// Mitsubishi GX Works2 project: Bread   PLC: FX3G

// global labels: Global1
VAR_GLOBAL
  Emergency AT X007 : BOOL;
  InputSpice AT M4 : BOOL;
  InputOil AT M3 : BOOL;
  InputWater AT M2 : BOOL;
  InputShmarim AT M1 : BOOL;
  InputYeast AT M1 : BOOL;
  InputFlour AT M0 : BOOL;
  StateEmergency AT M100 : BOOL;
  ReadyToStart AT Y000 : BOOL;
  StartDay AT X010 : BOOL;
  DayInProgress AT Y010 : BOOL;
  GetInput AT X000 : BOOL;
  AnalogInput1 AT D8280 : INT;
  FlourInStock AT D1101 : REAL;
END_VAR
VAR_GLOBAL CONSTANT
  Flour_Const : REAL := 100;
END_VAR
VAR_GLOBAL
  YeastInStock AT D1103 : REAL;
END_VAR
VAR_GLOBAL CONSTANT
  YeastRatio_Constant : REAL := 0.2;
END_VAR
VAR_GLOBAL
  WaterInStock AT D1105 : REAL;
END_VAR
VAR_GLOBAL CONSTANT
  WatertRatio_Constant : REAL := 0.5;
END_VAR
VAR_GLOBAL
  OilInStock AT D1107 : REAL;
END_VAR
VAR_GLOBAL CONSTANT
  OilRatio_Constant : REAL := 0.3;
END_VAR
VAR_GLOBAL
  SpiceInStock AT D1109 : REAL;
END_VAR
VAR_GLOBAL CONSTANT
  SpiceRatio_Constant : REAL := 0.1;
  Zero_Constant : REAL;
END_VAR
VAR_GLOBAL
  Lisha AT X001 : BOOL;
  Fiktivy AT M200 : BOOL;
  RealNura AT TC1 : BOOL;
END_VAR
VAR_GLOBAL CONSTANT
  mili_900 : INT := 4;
END_VAR
VAR_GLOBAL
  RealNuraTime AT TS1 : BOOL;
  FiktivylNura AT TC2 : BOOL;
END_VAR
VAR_GLOBAL CONSTANT
  mili_100 : INT := 1;
END_VAR
VAR_GLOBAL
  FiktivyNuraTime AT TS2 : BOOL;
  Fiktivy1 AT M300 : BOOL;
  NuraY0 AT M250 : BOOL;
  NuraDay AT M240 : BOOL;
  Emergency_ThreeSeconds AT TC3 : BOOL;
END_VAR
VAR_GLOBAL CONSTANT
  ThreeSeconds : INT := 30;
END_VAR
VAR_GLOBAL
  Emergency_ThreeSeconds_Time AT TS3 : BOOL;
END_VAR
VAR_GLOBAL CONSTANT
  mili_400 : INT := 4;
END_VAR
VAR_GLOBAL
  StartPrepare AT X002 : BOOL;
  Prepare_C AT TC30 : BOOL;
END_VAR
VAR_GLOBAL CONSTANT
  Prepare_milli : INT := 30;
END_VAR
VAR_GLOBAL
  StatePrepare AT M10 : BOOL;
  Prepare_Timer AT TS30 : BOOL;
  PrepareNura AT Y005 : BOOL;
  FinishPrepare AT M11 : BOOL;
  Flour_Mearbel AT D2101 : REAL;
  Yeast_Mearbel AT D2103 : REAL;
END_VAR
VAR_GLOBAL CONSTANT
  Yeast_Const : REAL := 20;
END_VAR
VAR_GLOBAL
  Flour_Meychal AT D2101 : REAL;
  Yeast_Meychal AT D2103 : REAL;
  Water_Meychal AT D2105 : REAL;
  Oil_Meychal AT D2107 : REAL;
END_VAR
VAR_GLOBAL CONSTANT
  Water_Const : REAL := 50;
  Oil_Const : REAL := 30;
  Spice_Const : REAL := 10;
END_VAR
VAR_GLOBAL
  Spice_Meychal AT D2109 : REAL;
  LishaNura AT Y001 : BOOL;
  Spice_Stock AT D1109 : REAL;
  StartHatfahaCount AT CC0 : BOOL;
END_VAR
VAR_GLOBAL CONSTANT
  count2 : INT := 2;
END_VAR
VAR_GLOBAL
  StartHatfaha AT CS0 : BOOL;
  FakeNuraY1 AT M252 : BOOL;
  NuraY2 AT Y002 : BOOL;
  NuraY3 AT Y003 : BOOL;
  Y2NuraTime AT TS10 : BOOL;
  Y3NuraTime AT TS20 : BOOL;
  Hatfaha_ThreeSeconds_Time AT TS80 : BOOL;
  HivHov AT M280 : BOOL;
  HivHovY2 AT TC10 : BOOL;
  HivHovY3 AT TC20 : BOOL;
  Hatfaha_ThreeSeconds AT TC80 : BOOL;
  StartHivHov AT M80 : BOOL;
  Hatfaha_Tavnit AT D4101 : REAL;
END_VAR
VAR_GLOBAL CONSTANT
  Batzekr_Const : REAL := 210;
  Batzek_Const : REAL := 210;
  Afia_time_const : WORD := 40;
END_VAR
VAR_GLOBAL
  NuraY4 AT TC90 : BOOL;
  Hatfaha AT X011 : BOOL;
  Lisha_mearbelNEW AT D3101 : REAL;
  Afia_done AT TS90 : BOOL;
  NuraAfiaY4 AT Y004 : BOOL;
  bdika AT X005 : BOOL;
  bdikanura AT Y011 : BOOL;
  end_hatfaha AT M244 : BOOL;
  StartQA AT X003 : BOOL;
  QA_input AT D5101 : REAL;
END_VAR
VAR_GLOBAL CONSTANT
  QA_const_1 : INT := 400;
  QA_const_5 : INT := 2000;
END_VAR
VAR_GLOBAL
  QA_Success AT M197 : BOOL;
  NuraY6 AT TC95 : BOOL;
END_VAR
VAR_GLOBAL CONSTANT
  shelf_tranfer_time : WORD := 50;
END_VAR
VAR_GLOBAL
  Shelf_transfer_done AT TS95 : BOOL;
  NuraY5 AT Y005 : BOOL;
END_VAR
VAR_GLOBAL CONSTANT
  count_QA_CONST : INT := 2;
END_VAR
VAR_GLOBAL
  count_QA AT CC2 : BOOL;
  count_QA_done AT CS2 : BOOL;
  Afia_tavnit AT D6101 : REAL;
  Fiktivi_QA_succes AT M325 : BOOL;
  Bread_shelf AT D7101 : REAL;
  Greater_than1 AT M222 : BOOL;
  Less_than5 AT M223 : BOOL;
  QA_Success_NuraY6 AT Y006 : BOOL;
  Input_saved AT M127 : BOOL;
  AnalogInput2 AT D8281 : INT;
  AnalogOutput AT D8201 : INT;
  Ingridients_check AT M255 : BOOL;
  AnalogOutputnEW AT D8201 : INT;
  StartHatfaha_current AT CN0 : INT;
  count_QA_current AT CN2 : INT;
END_VAR
VAR_GLOBAL CONSTANT
  Zero_Constant_Word : INT;
END_VAR
VAR_GLOBAL
  Ge_success AT M190 : BOOL;
  Le_success AT M191 : BOOL;
  checkIngridients AT M321 : BOOL;
END_VAR

// task Task_01 (event TRUE, interval 0, priority 31): POU_01

PROGRAM POU_01
VAR
  Lisha_mearbel : REAL;
END_VAR
(* structured ladder/FBD written out as ST: instructions are called as NAME(EN, inputs, outputs); _pN, _eN, _tN stand for wires *)
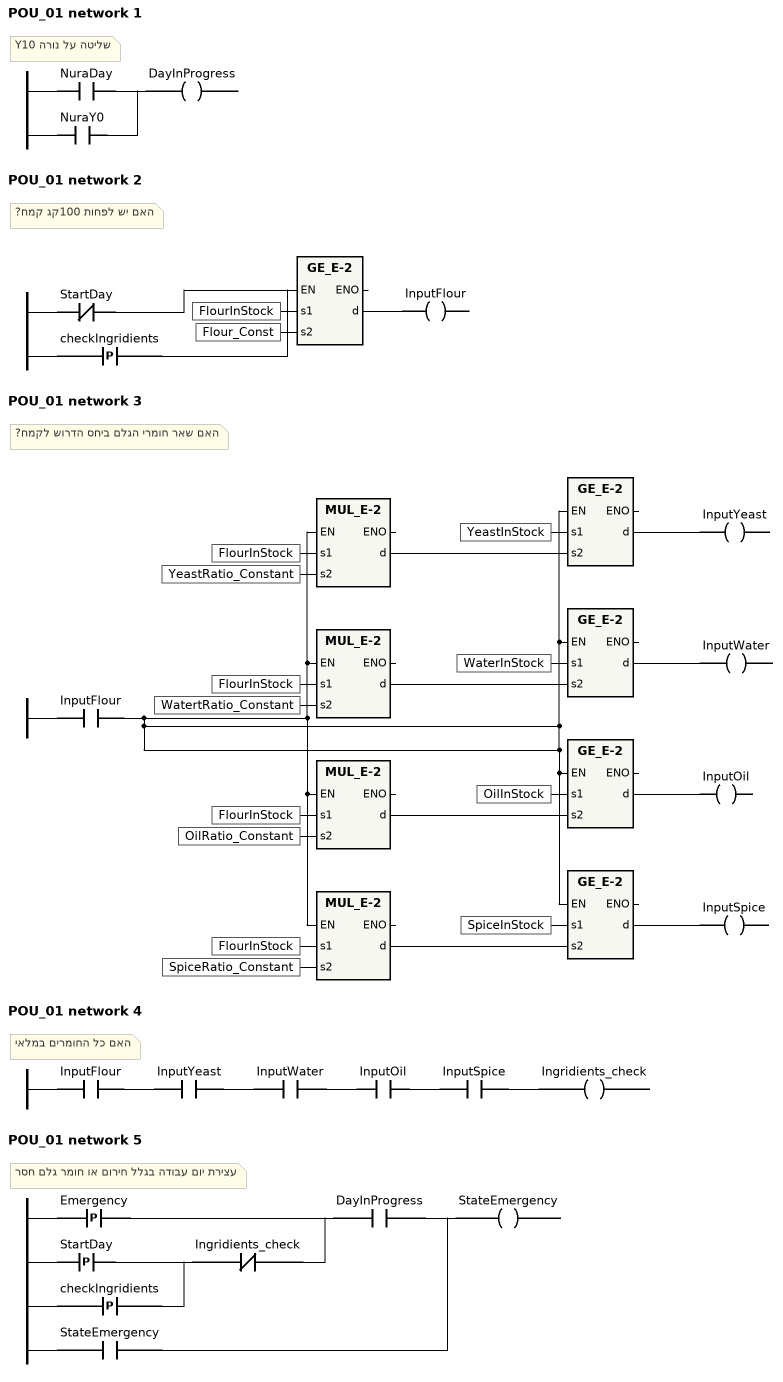
(* network 1 *)
(* שליטה על נורה Y10 *)
DayInProgress := NuraDay OR NuraY0;
(* network 2 *)
(* האם יש לפחות 100קג קמח? *)
GE_E((NOT StartDay) OR LDP(TRUE, checkIngridients), FlourInStock, Flour_Const, _t1);
InputFlour := _t1;
(* network 3 *)
(* האם שאר חומרי הגלם ביחס הדרוש לקמח? *)
MUL_E(InputFlour, FlourInStock, YeastRatio_Constant, _t1);
GE_E(InputFlour, YeastInStock, _t1, _t2);
InputYeast := _t2;
MUL_E(InputFlour, FlourInStock, WatertRatio_Constant, _t3);
GE_E(InputFlour, WaterInStock, _t3, _t4);
InputWater := _t4;
MUL_E(InputFlour, FlourInStock, OilRatio_Constant, _t5);
GE_E(InputFlour, OilInStock, _t5, _t6);
InputOil := _t6;
MUL_E(InputFlour, FlourInStock, SpiceRatio_Constant, _t7);
GE_E(InputFlour, SpiceInStock, _t7, _t8);
InputSpice := _t8;
(* network 4 *)
(* האם כל החומרים במלאי *)
Ingridients_check := InputFlour AND InputYeast AND InputWater AND InputOil AND InputSpice;
(* network 5 *)
(* עצירת יום עבודה בגלל חירום או חומר גלם חסר *)
StateEmergency := ((LDP(TRUE, Emergency) OR ((LDP(TRUE, StartDay) OR LDP(TRUE, checkIngridients)) AND NOT Ingridients_check)) AND DayInProgress) OR StateEmergency;
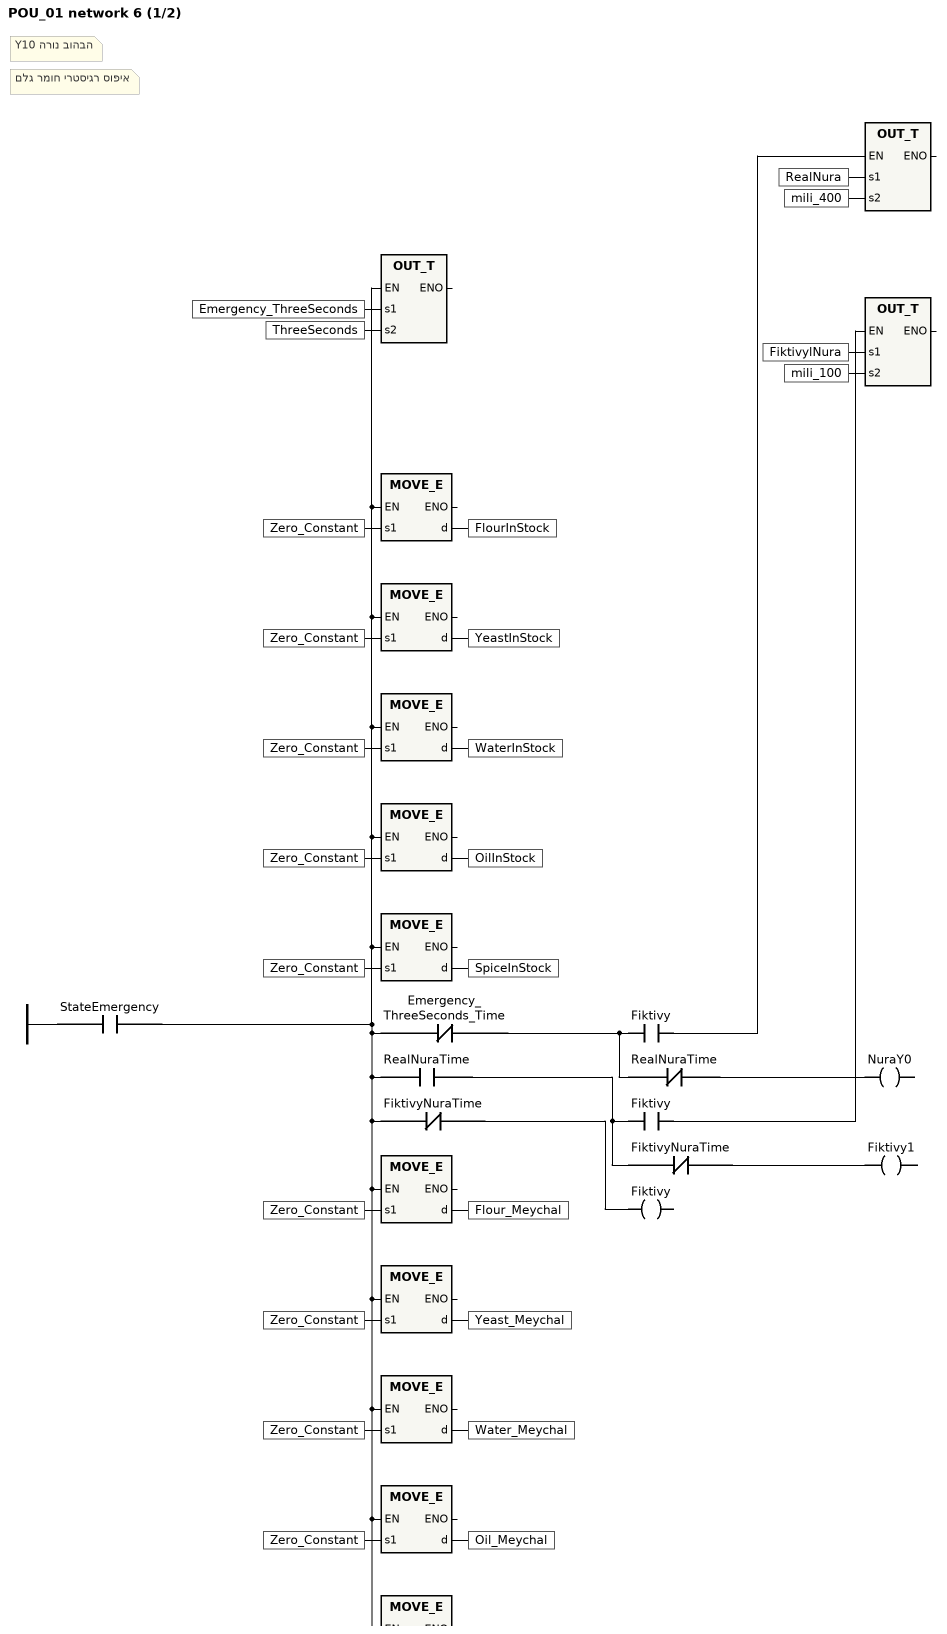
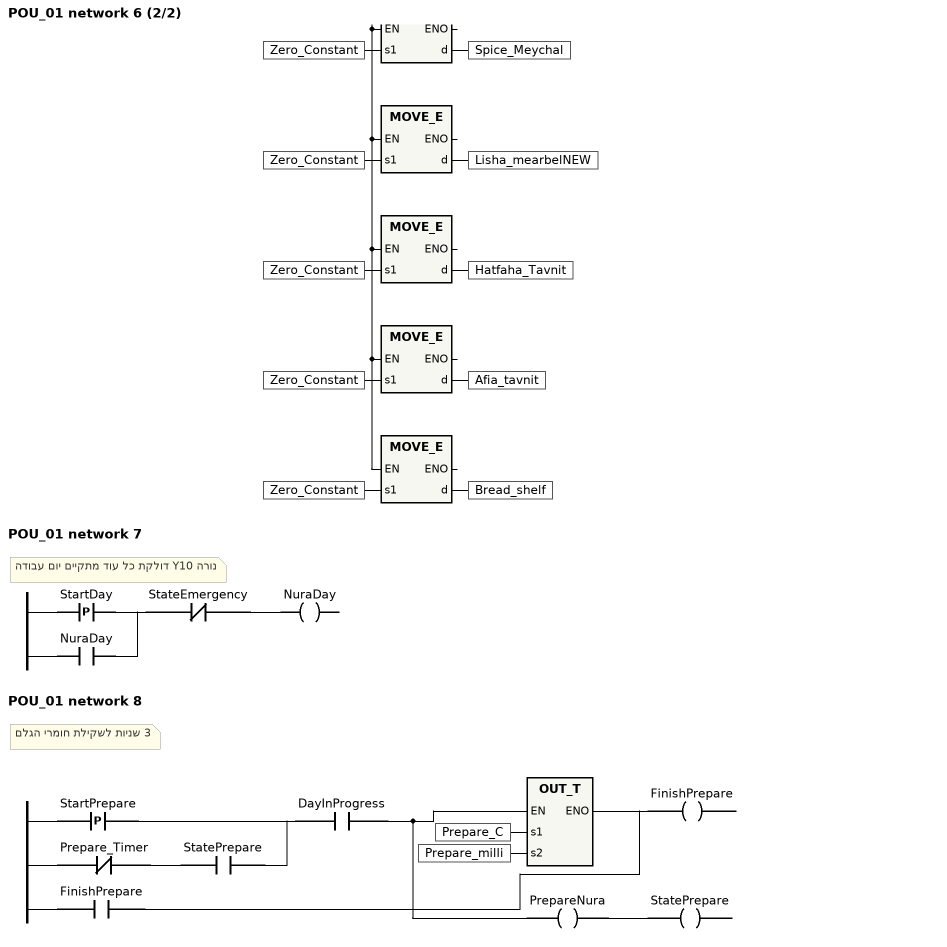
(* network 6 *)
(* הבהוב נורה Y10 *)
(* איפוס רגיסטרי חומר גלם *)
_p1 := StateEmergency AND NOT Emergency_ThreeSeconds_Time;
OUT_T(_p1 AND Fiktivy, RealNura, mili_400);
NuraY0 := _p1 AND NOT RealNuraTime;
_p2 := StateEmergency AND RealNuraTime;
OUT_T(_p2 AND Fiktivy, FiktivylNura, mili_100);
Fiktivy1 := _p2 AND NOT FiktivyNuraTime;
Fiktivy := StateEmergency AND NOT FiktivyNuraTime;
OUT_T(StateEmergency, Emergency_ThreeSeconds, ThreeSeconds);
MOVE_E(StateEmergency, Zero_Constant, FlourInStock);
MOVE_E(StateEmergency, Zero_Constant, YeastInStock);
MOVE_E(StateEmergency, Zero_Constant, WaterInStock);
MOVE_E(StateEmergency, Zero_Constant, OilInStock);
MOVE_E(StateEmergency, Zero_Constant, SpiceInStock);
MOVE_E(StateEmergency, Zero_Constant, Flour_Meychal);
MOVE_E(StateEmergency, Zero_Constant, Yeast_Meychal);
MOVE_E(StateEmergency, Zero_Constant, Water_Meychal);
MOVE_E(StateEmergency, Zero_Constant, Oil_Meychal);
MOVE_E(StateEmergency, Zero_Constant, Spice_Meychal);
MOVE_E(StateEmergency, Zero_Constant, Lisha_mearbelNEW);
MOVE_E(StateEmergency, Zero_Constant, Hatfaha_Tavnit);
MOVE_E(StateEmergency, Zero_Constant, Afia_tavnit);
MOVE_E(StateEmergency, Zero_Constant, Bread_shelf);
(* network 7 *)
(* נורה Y10 דולקת כל עוד מתקיים יום עבודה *)
NuraDay := (LDP(TRUE, StartDay) OR NuraDay) AND NOT StateEmergency;
(* network 8 *)
(* 3 שניות לשקילת חומרי הגלם *)
_p1 := (LDP(TRUE, StartPrepare) OR (NOT Prepare_Timer AND StatePrepare)) AND DayInProgress;
PrepareNura := _p1;
StatePrepare := _p1;
_e2 := OUT_T(_p1, Prepare_C, Prepare_milli);
FinishPrepare := _e2 OR FinishPrepare;
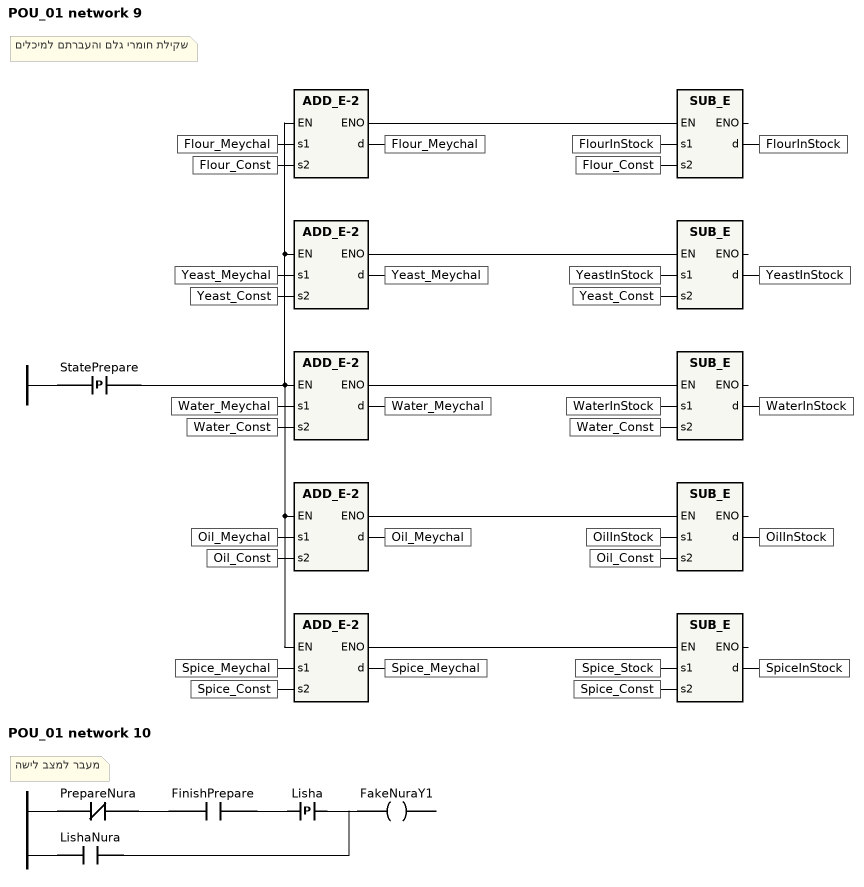
(* network 9 *)
(* שקילת חומרי גלם והעברתם למיכלים *)
_p1 := LDP(TRUE, StatePrepare);
_e2 := ADD_E(_p1, Flour_Meychal, Flour_Const, Flour_Meychal);
SUB_E(_e2, FlourInStock, Flour_Const, FlourInStock);
_e3 := ADD_E(_p1, Yeast_Meychal, Yeast_Const, Yeast_Meychal);
SUB_E(_e3, YeastInStock, Yeast_Const, YeastInStock);
_e4 := ADD_E(_p1, Water_Meychal, Water_Const, Water_Meychal);
SUB_E(_e4, WaterInStock, Water_Const, WaterInStock);
_e5 := ADD_E(_p1, Oil_Meychal, Oil_Const, Oil_Meychal);
SUB_E(_e5, OilInStock, Oil_Const, OilInStock);
_e6 := ADD_E(_p1, Spice_Meychal, Spice_Const, Spice_Meychal);
SUB_E(_e6, Spice_Stock, Spice_Const, SpiceInStock);
(* network 10 *)
(* מעבר למצב לישה *)
FakeNuraY1 := (NOT PrepareNura AND FinishPrepare AND LDP(TRUE, Lisha)) OR LishaNura;
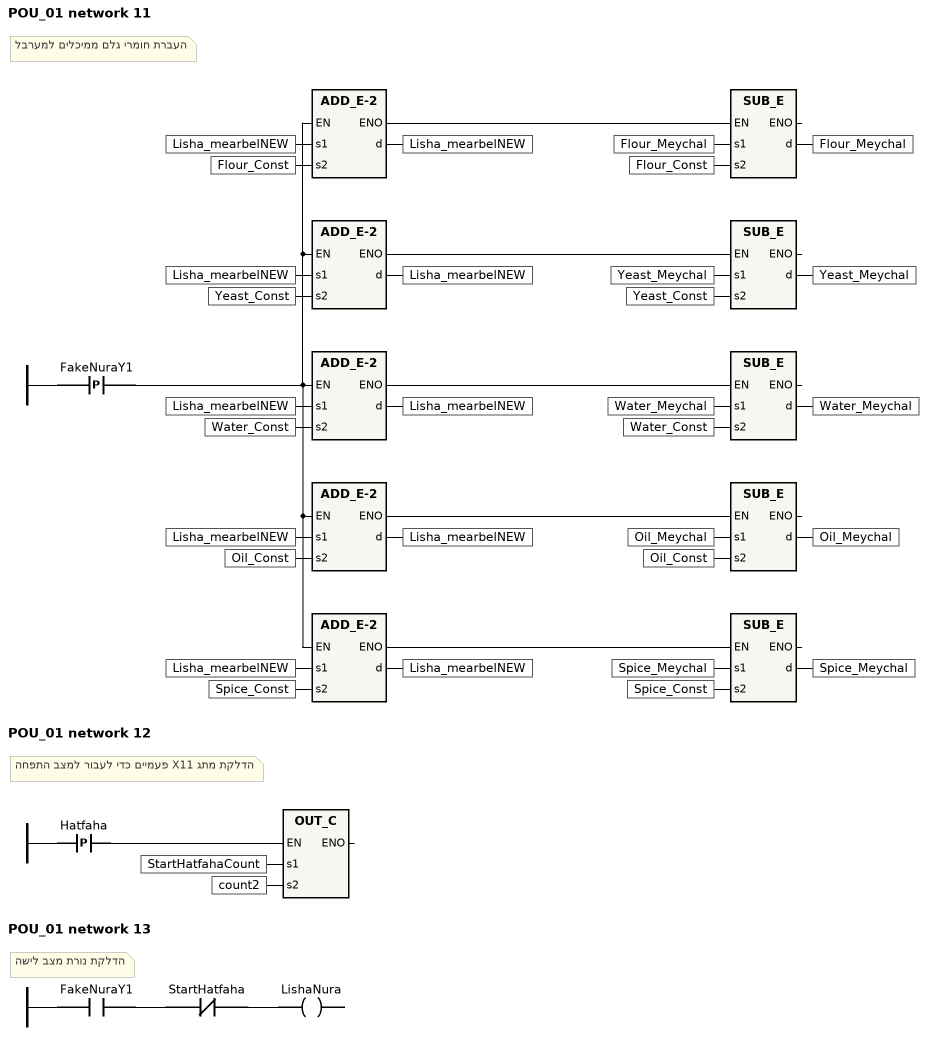
(* network 11 *)
(* העברת חומרי גלם ממיכלים למערבל *)
_p1 := LDP(TRUE, FakeNuraY1);
_e2 := ADD_E(_p1, Lisha_mearbelNEW, Flour_Const, Lisha_mearbelNEW);
SUB_E(_e2, Flour_Meychal, Flour_Const, Flour_Meychal);
_e3 := ADD_E(_p1, Lisha_mearbelNEW, Yeast_Const, Lisha_mearbelNEW);
SUB_E(_e3, Yeast_Meychal, Yeast_Const, Yeast_Meychal);
_e4 := ADD_E(_p1, Lisha_mearbelNEW, Water_Const, Lisha_mearbelNEW);
SUB_E(_e4, Water_Meychal, Water_Const, Water_Meychal);
_e5 := ADD_E(_p1, Lisha_mearbelNEW, Oil_Const, Lisha_mearbelNEW);
SUB_E(_e5, Oil_Meychal, Oil_Const, Oil_Meychal);
_e6 := ADD_E(_p1, Lisha_mearbelNEW, Spice_Const, Lisha_mearbelNEW);
SUB_E(_e6, Spice_Meychal, Spice_Const, Spice_Meychal);
(* network 12 *)
(* הדלקת מתג X11 פעמיים כדי לעבור למצב התפחה *)
OUT_C(LDP(TRUE, Hatfaha), StartHatfahaCount, count2);
(* network 13 *)
(* הדלקת נורת מצב לישה *)
LishaNura := FakeNuraY1 AND NOT StartHatfaha;
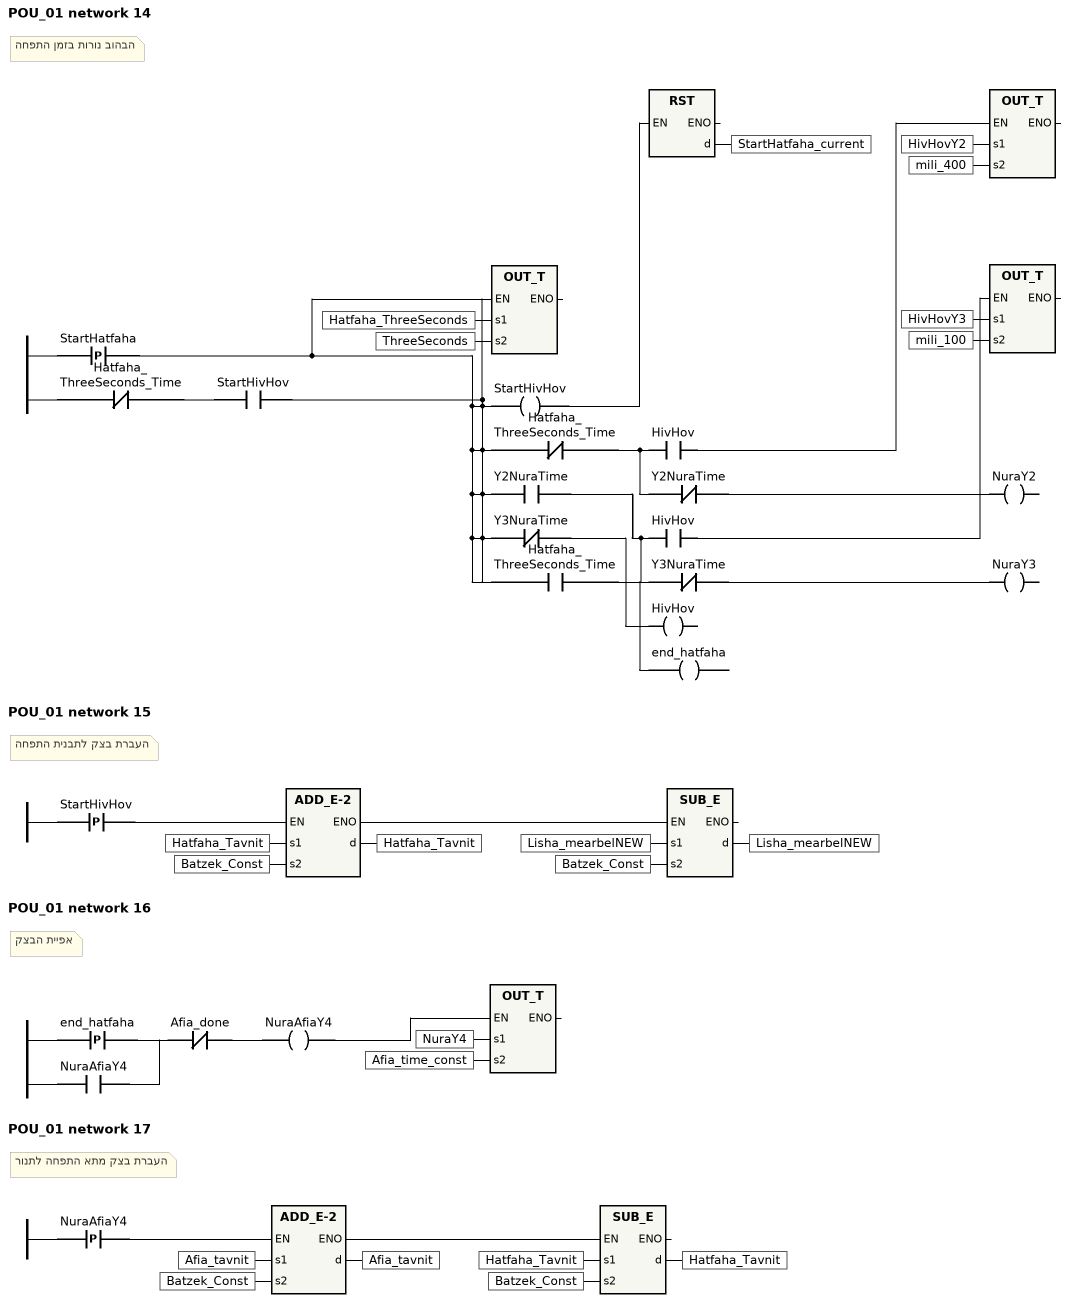
(* network 14 *)
(* הבהוב נורות בזמן התפחה *)
_p1 := LDP(TRUE, StartHatfaha) OR (NOT Hatfaha_ThreeSeconds_Time AND StartHivHov);
StartHivHov := _p1;
RST(_p1, StartHatfaha_current);
_p2 := _p1 AND NOT Hatfaha_ThreeSeconds_Time;
OUT_T(_p2 AND HivHov, HivHovY2, mili_400);
NuraY2 := _p2 AND NOT Y2NuraTime;
_p3 := _p1 AND Y2NuraTime;
OUT_T(_p3 AND HivHov, HivHovY3, mili_100);
NuraY3 := _p3 AND NOT Y3NuraTime;
HivHov := _p1 AND NOT Y3NuraTime;
OUT_T(_p1, Hatfaha_ThreeSeconds, ThreeSeconds);
end_hatfaha := _p1 AND Hatfaha_ThreeSeconds_Time;
(* network 15 *)
(* העברת בצק לתבנית התפחה *)
_e1 := ADD_E(LDP(TRUE, StartHivHov), Hatfaha_Tavnit, Batzek_Const, Hatfaha_Tavnit);
SUB_E(_e1, Lisha_mearbelNEW, Batzek_Const, Lisha_mearbelNEW);
(* network 16 *)
(* אפיית הבצק *)
_p1 := (LDP(TRUE, end_hatfaha) OR NuraAfiaY4) AND NOT Afia_done;
NuraAfiaY4 := _p1;
OUT_T(_p1, NuraY4, Afia_time_const);
(* network 17 *)
(* העברת בצק מתא התפחה לתנור *)
_e1 := ADD_E(LDP(TRUE, NuraAfiaY4), Afia_tavnit, Batzek_Const, Afia_tavnit);
SUB_E(_e1, Hatfaha_Tavnit, Batzek_Const, Hatfaha_Tavnit);
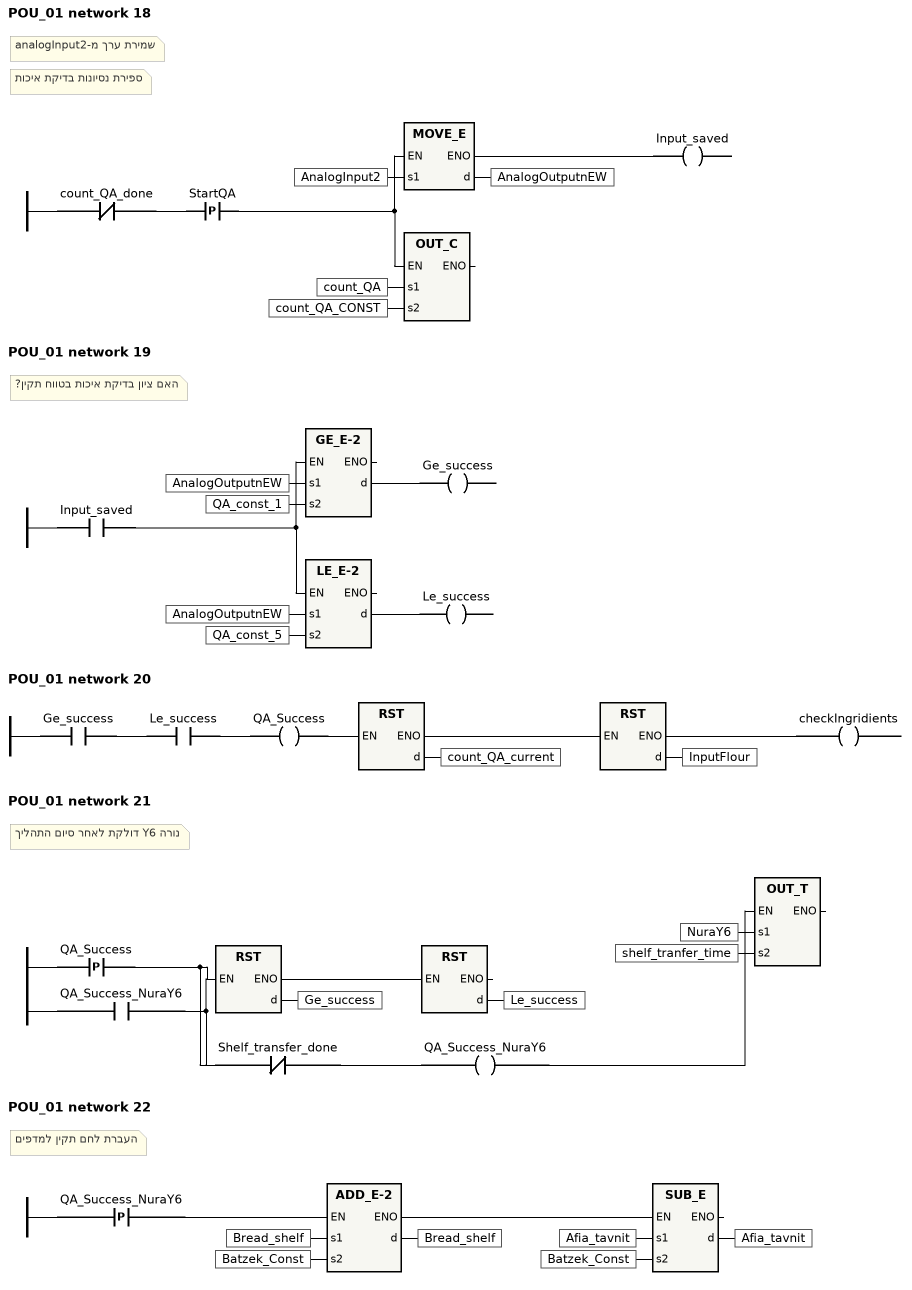
(* network 18 *)
(* שמירת ערך מ-analogInput2 *)
(* ספירת נסיונות בדיקת איכות *)
_p1 := NOT count_QA_done AND LDP(TRUE, StartQA);
_e2 := MOVE_E(_p1, AnalogInput2, AnalogOutputnEW);
Input_saved := _e2;
OUT_C(_p1, count_QA, count_QA_CONST);
(* network 19 *)
(* האם ציון בדיקת איכות בטווח תקין? *)
GE_E(Input_saved, AnalogOutputnEW, QA_const_1, _t1);
Ge_success := _t1;
LE_E(Input_saved, AnalogOutputnEW, QA_const_5, _t2);
Le_success := _t2;
(* network 20 *)
_p1 := Ge_success AND Le_success;
QA_Success := _p1;
_e2 := RST(_p1, count_QA_current);
_e3 := RST(_e2, InputFlour);
checkIngridients := _e3;
(* network 21 *)
(* נורה Y6 דולקת לאחר סיום התהליך *)
_p1 := LDP(TRUE, QA_Success) OR QA_Success_NuraY6;
_p2 := _p1 AND NOT Shelf_transfer_done;
QA_Success_NuraY6 := _p2;
OUT_T(_p2, NuraY6, shelf_tranfer_time);
_e3 := RST(_p1, Ge_success);
RST(_e3, Le_success);
(* network 22 *)
(* העברת לחם תקין למדפים *)
_e1 := ADD_E(LDP(TRUE, QA_Success_NuraY6), Bread_shelf, Batzek_Const, Bread_shelf);
SUB_E(_e1, Afia_tavnit, Batzek_Const, Afia_tavnit);
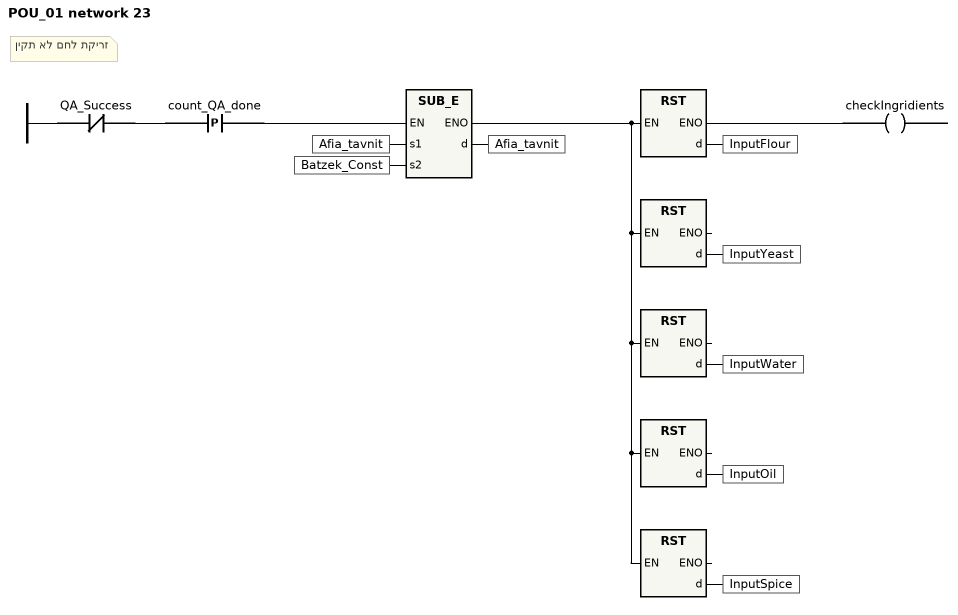
(* network 23 *)
(* זריקת לחם לא תקין *)
_e1 := SUB_E(NOT QA_Success AND LDP(TRUE, count_QA_done), Afia_tavnit, Batzek_Const, Afia_tavnit);
_e2 := RST(_e1, InputFlour);
checkIngridients := _e2;
RST(_e1, InputYeast);
RST(_e1, InputWater);
RST(_e1, InputOil);
RST(_e1, InputSpice);
END_PROGRAM
